FUNCTION_BLOCK FB_SXR_SATT_Stage
VAR_IN_OUT
    stAxis : DUT_MotionStage;
END_VAR
VAR_INPUT
    nEnableMode : ENUM_StageEnableMode;
END_VAR
VAR_OUTPUT
END_VAR
VAR
    // TODO: debug
    // fbMotion: FB_MotionStage;
    fbMotion: FB_MotionStageSim;

    stExtra : DUT_MotionStage_Extras;
    bInitialized: BOOL := FALSE;
END_VAR

IF bInitialized THEN
    bInitialized := TRUE;

    (* Defaults for DUT_MotionStage *)
    stAxis.bHardwareEnable      := TRUE;
    stAxis.bLimitBackwardEnable := TRUE;
    stAxis.bLimitForwardEnable  := TRUE;
    stAxis.bPowerSelf           := TRUE;
    stAxis.nBrakeMode           := ENUM_StageBrakeMode.NO_BRAKE;
    stAxis.nHomingMode          := ENUM_EpicsHomeCmd.NONE;

    (* Defaults for visualization *)
    stExtra.fVisuStep			:= 0.1;

END_IF

stAxis.nEnableMode := nEnableMode;
fbMotion(stMotionStage:=stAxis);

stExtra.bVisuHighLim := NOT stAxis.bAllForwardEnable;
stExtra.bVisuLowLim := NOT stAxis.bAllBackwardEnable;

END_FUNCTION_BLOCK

(* stored: Version 1.1.0.1, ProductVersion 3.1.4024.4
   POU FB_SXR_SATT_Stage: Id {7fb611c7-2215-4e8f-8a28-e51a98acae9a}, SpecialFunc None *)
